// Mitsubishi GX Works2 project: timer3   PLC: Q03UDV

PROGRAM MAIN
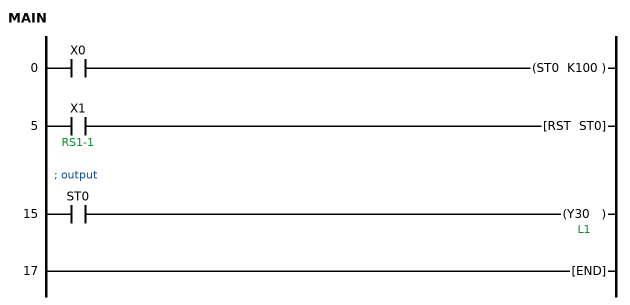
0     LD      X0
      OUT     ST0 K100
5     LD      X1  ; RS1-1
      RST     ST0
; output
15    LD      ST0
      OUT     Y30  ; L1
17    END
END_PROGRAM

// device comments not shown above
X2  ; RS1-2
X3  ; RS2-1
X4  ; RS2-2
X15  ; PB1
X16  ; PB2
X17  ; PB3
X18  ; PB4
X19  ; PB5
X1A  ; PB6
X1B  ; PB7
X1C  ; PB8
Y31  ; L2
Y32  ; L3
Y33  ; L4
Y34  ; L5
Y35  ; L6
Y36  ; L7
Y38  ; SV1-1
Y39  ; SV1-2
Y3A  ; SV2
Y3B  ; SV3
